SUBAPPLICATION Uebung_029 (* LED_DO Blinkende LED *)
  (* Standard: 61499-2; Description: Copyright (c) 2023 Meisterschulen am Ostbahnhof This program and the accompanying materials are made available under the terms of the Eclipse Public License 2.0 which is available at https://www.eclipse.org/legal/epl-2.0/ SPDX-License-Identifier: EPL-2.0 *)
  (* Version 1.0, 2023-10-23, Franz Höpfinger, Meisterschulen am Ostbahnhof *)
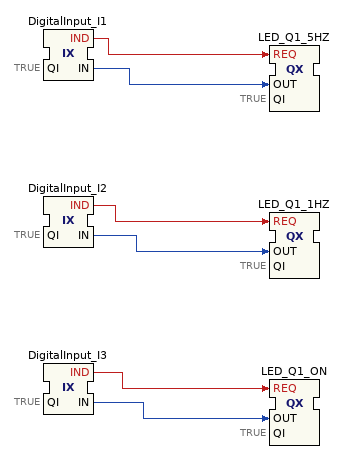
  FBS
    LED_Q1_5HZ : QX(QI := TRUE);
    DigitalInput_I1 : IX(QI := TRUE);
    LED_Q1_1HZ : QX(QI := TRUE);
    DigitalInput_I2 : IX(QI := TRUE);
    LED_Q1_ON : QX(QI := TRUE);
    DigitalInput_I3 : IX(QI := TRUE);
  END_FBS
  EVENT_CONNECTIONS
    DigitalInput_I1.IND TO LED_Q1_5HZ.REQ;
    DigitalInput_I2.IND TO LED_Q1_1HZ.REQ;
    DigitalInput_I3.IND TO LED_Q1_ON.REQ;
  END_CONNECTIONS
  DATA_CONNECTIONS
    DigitalInput_I1.IN TO LED_Q1_5HZ.OUT;
    DigitalInput_I2.IN TO LED_Q1_1HZ.OUT;
    DigitalInput_I3.IN TO LED_Q1_ON.OUT;
  END_CONNECTIONS
END_SUBAPPLICATION
